Fanuc KAREL source: KT00649.KL

PROGRAM KT00649
%NOLOCKGROUP
VAR
  H1: ARRAY[2] OF SHORT
  H2: ARRAY[2] OF SHORT
  OUT: INTEGER
BEGIN
  H1[1] = 2
  H2[1] = 3
  H1[1] = 2
  H2[1] = 3
  OUT = - H1[1]
END KT00649
